FUNCTION_BLOCK TIMESERIES_CORRELATION_ANALYSIS
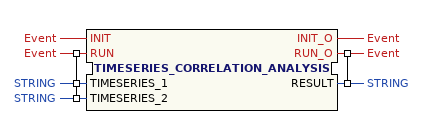
  EVENT_INPUT
    INIT;
    RUN WITH TIMESERIES_1, TIMESERIES_2;
  END_EVENT
  EVENT_OUTPUT
    INIT_O;
    RUN_O WITH RESULT;
  END_EVENT
  VAR_INPUT
    TIMESERIES_1 : STRING;
    TIMESERIES_2 : STRING;
  END_VAR
  VAR_OUTPUT
    RESULT : STRING;
  END_VAR
END_FUNCTION_BLOCK
